// TwinCAT 3 PLC project TcMath
// ProgramVersion: 3.1.4022.4
// libraries:
//   Tc2_Standard, * (Beckhoff Automation GmbH)
//   Tc2_System, * (Beckhoff Automation GmbH)
//   Tc3_Module, * (Beckhoff Automation GmbH)
//   TcUnit, * (www.tcunit.org)
// project tree:
//   / PlcTask.TcTTO
//   POUs/ FB_MovingAverage.TcPOU
//   Test/ FB_MovingAverage_Test.TcPOU, PRG_TEST.TcPOU
// real-time tasks:
//   TASK PlcTask: cycle T#10ms, priority 20, ADS port 350

CONFIGURATION TcMath
    RESOURCE PLC ON TwinCAT3
        TASK PlcTask(INTERVAL := T#10ms, PRIORITY := 20);
        PROGRAM PRG_TEST WITH PlcTask : PRG_TEST;
    END_RESOURCE
END_CONFIGURATION

// ---- Test/PRG_TEST.TcPOU
PROGRAM PRG_TEST
VAR
    MovingAverage_Test : FB_MovingAverage_Test;
END_VAR

TcUnit.RUN();

END_PROGRAM

// ---- Test/FB_MovingAverage_Test.TcPOU
{attribute 'call_after_init'}
FUNCTION_BLOCK FB_MovingAverage_Test EXTENDS FB_TestSuite IMPLEMENTS I_RunnableTestSuite
VAR
    Assert : TcUnit.FB_Assert;
END_VAR

METHOD PRIVATE AddFiveNumbersExpectAverageOfAll
VAR
    DataArray : ARRAY[1..5] OF LREAL;
    MovingAverage : FB_MovingAverage(StorageArray := ADR(DataArray), FilterSize := 5);

    ExpectedValue : LREAL := 1.0;
    CurrentAverage : LREAL;
END_VAR
TEST('AddFiveNumbersExpectAverageOfAll');

MovingAverage.AddDataPoint(x := 1.0);
MovingAverage.AddDataPoint(x := 1.0);
MovingAverage.AddDataPoint(x := 1.0);
MovingAverage.AddDataPoint(x := 1.0);
MovingAverage.AddDataPoint(x := 1.0);

CurrentAverage := MovingAverage.GetAverage();

Assert.AssertEquals(Expected := ExpectedValue,
                    Actual := CurrentAverage,
                    Message := 'Moving average value not correct');
END_METHOD

METHOD PRIVATE AddJustOneNumberExpectAverageToBeThatOneNumber
VAR
    DataArray : ARRAY[0..4] OF LREAL;
    MovingAverage : FB_MovingAverage(StorageArray := ADR(DataArray), FilterSize := 5);
    ExpectedValue : LREAL := 113.0;
    CurrentAverage : LREAL;
END_VAR
TEST('AddJustOneNumberExpectAverageToBeThatOneNumber');

MovingAverage.AddDataPoint(x := 113.0);

CurrentAverage := MovingAverage.GetAverage();

Assert.AssertEquals(Expected := ExpectedValue,
                    Actual := CurrentAverage,
                    Message := 'Moving average value not correct');
END_METHOD

METHOD PRIVATE AddLessThanFilterSizeExpectAverageOfAddedValues
VAR
    DataArray : ARRAY[1..5] OF LREAL;
    MovingAverage : FB_MovingAverage(StorageArray := ADR(DataArray), FilterSize := 5);
END_VAR
TEST('AddLessThanFilterSizeExpectAverageOfAddedValues');

MovingAverage.AddDataPoint(x := 110.0);
MovingAverage.AddDataPoint(x := 5.0);

Assert.AssertEquals_LREAL(Expected := 57.5,
                          Actual := MovingAverage.GetAverage(),
                          Delta := 0.0001,
                          Message := 'Moving average value not correct');
END_METHOD

METHOD PRIVATE AddMoreThanFilterSizeExpectAverageOfLastAdded
VAR
    DataArray : ARRAY[4..6] OF LREAL;
    MovingAverage : FB_MovingAverage(StorageArray := ADR(DataArray), FilterSize := 3);

    ExpectedValue : LREAL := 115.74292;
    CurrentAverage : LREAL;
END_VAR
TEST('AddMoreThanFilterSizeExpectAverageOfLastAdded');

MovingAverage.AddDataPoint(x := 4.5135);
MovingAverage.AddDataPoint(x := 84.76436);
MovingAverage.AddDataPoint(x := 257.123);
MovingAverage.AddDataPoint(x := 5.3414);

Assert.AssertEquals_LREAL(Expected := 115.74292,
                          Actual := MovingAverage.GetAverage(),
                          Delta := 0.01,
                          Message := 'Moving average value not correct');
END_METHOD

METHOD FB_init : BOOL
VAR_INPUT
	bInitRetains : BOOL; // if TRUE, the retain variables are initialized (warm start / cold start)
	bInCopyCode : BOOL;  // if TRUE, the instance afterwards gets moved into the copy code (online change)
END_VAR
SUPER^.RegisterTestSuite(THIS^);
END_METHOD

METHOD RunTests : TCUNIT.E_TestSuiteRunState
AddFiveNumbersExpectAverageOfAll();
AddLessThanFilterSizeExpectAverageOfAddedValues();
UseBiggerStorageThanFilterSizeExpectAverageOfFilterSize();
AddMoreThanFilterSizeExpectAverageOfLastAdded();
AddJustOneNumberExpectAverageToBeThatOneNumber();

RunTests := TCUNIT.E_TestSuiteRunState.FINISHED;
END_METHOD

METHOD PRIVATE UseBiggerStorageThanFilterSizeExpectAverageOfFilterSize
VAR
    DataArray : ARRAY[1..5] OF LREAL;
    MovingAverage : FB_MovingAverage(StorageArray := ADR(DataArray), FilterSize := 3);

    ExpectedValue : LREAL := 11.0;
    CurrentAverage : LREAL;
END_VAR
TEST('UseBiggerStorageThanFilterSizeExpectAverageOfFilterSize');

MovingAverage.AddDataPoint(x := 2.0);
MovingAverage.AddDataPoint(x := 3.0);
MovingAverage.AddDataPoint(x := 4.0);
MovingAverage.AddDataPoint(x := 5.0);
MovingAverage.AddDataPoint(x := 6.0);
MovingAverage.AddDataPoint(x := 7.0);
MovingAverage.AddDataPoint(x := 8.0);
MovingAverage.AddDataPoint(x := 9.0);
MovingAverage.AddDataPoint(x := 10.0);
MovingAverage.AddDataPoint(x := 11.0);
MovingAverage.AddDataPoint(x := 12.0);

CurrentAverage := MovingAverage.GetAverage();

Assert.AssertEquals(Expected := ExpectedValue,
                    Actual := CurrentAverage,
                    Message := 'Moving average value not correct');
END_METHOD

END_FUNCTION_BLOCK

// ---- POUs/FB_MovingAverage.TcPOU
FUNCTION_BLOCK FB_MovingAverage
VAR
    _StorageArray : POINTER TO LREAL;
    _FilterSize : UINT;

    Index : INT := -1;
    Average, Sum : LREAL;

    EqualOrMoreDataPointsThanFilterSize : BOOL := FALSE;
END_VAR

METHOD PUBLIC AddDataPoint
VAR_INPUT
    x : LREAL;
END_VAR
Index := (Index + 1) MOD UINT_TO_INT(_FilterSize);

Sum := Sum - _StorageArray[Index];
_StorageArray[Index] := x;
Sum := Sum + x;

IF NOT EqualOrMoreDataPointsThanFilterSize AND (Index = (UINT_TO_INT(_FilterSize) - 1)) THEN
    EqualOrMoreDataPointsThanFilterSize := TRUE;
END_IF

IF EqualOrMoreDataPointsThanFilterSize THEN
    Average := Sum / UINT_TO_LREAL(_FilterSize);
ELSE
    Average := Sum / INT_TO_LREAL(Index + 1);
END_IF
END_METHOD

METHOD FB_init : BOOL
VAR_INPUT
	bInitRetains : BOOL; // if TRUE, the retain variables are initialized (warm start / cold start)
	bInCopyCode : BOOL;  // if TRUE, the instance afterwards gets moved into the copy code (online change)
    StorageArray : POINTER TO LREAL;
    FilterSize : UINT;
END_VAR
_StorageArray := StorageArray;
_FilterSize := FilterSize;
END_METHOD

METHOD PUBLIC GetAverage : LREAL
GetAverage := Average;
END_METHOD

END_FUNCTION_BLOCK
